// TIA Portal V17 export
// export: Created 2023-12-22T15:08:07.2930648Z, ExportSetting WithDefaults, DisplayName Totally Integrated Automation Portal, DisplayVersion V17, DisplayName TIA Portal Openness, DisplayVersion V17, DisplayName TIA Portal Version Control Interface, DisplayVersion V17, DisplayName STEP 7 Professional, DisplayVersion V17, DisplayName STEP 7 Safety, DisplayVersion V17, DisplayName WinCC Advanced, DisplayVersion V17
FUNCTION_BLOCK "Time_SYS"   // FB95, LAD
{ S7_Optimized_Access := 'FALSE' }
VERSION : 0.1
// stored: AutoNumber false, IsIECCheckEnabled false, SetENOAutomatically false, UDAEnableTagReadback false
   VAR DB_SPECIFIC
      Set_Time : Bool;   // Заданное время
      Time_Now : Struct   // Текущее время
         Year : Int;   // год
         Month : Int;   // месяц
         Day : Int;   // день месяца
         Weekday : Int;   // день недели (1 - воскресенье)
         Hour : Int;   // часы
         Minute : Int;   // минуты
         Second : Int;   // секунды
      END_STRUCT;
      Time_SP : Struct   // Текущее время
         Year : Int;   // год
         Month : Int;   // месяц
         Day : Int;   // день месяца
         Weekday : Int;   // день недели (1 - воскресенье)
         Hour : Int;   // часы
         Minute : Int;   // минуты
         Second : Int;   // секунды
      END_STRUCT;
      TimeZone { S7_SetPoint := 'True'} : TimeTransformationRule;   // Часовой пояс
      RD_SYS_Status : Int;   // Статус чтения времени
      WR_SYS_Status : Int;   // Статус записи времени
      RD_Time : DTL;   // Прочитанное сист. время
      SP_Time : DTL;   // Новое сист. время
   END_VAR
   VAR
      SET_TIMEZONE { S7_SetPoint := 'True'} : SET_TIMEZONE;   // Запись часового пояса
   END_VAR
   VAR DB_SPECIFIC
      Time_DTL : DTL;
   END_VAR
   // TimeZone.Bias := 180;   // Часовой пояс по GMT (смещение в минутах)
   // TimeZone.DaylightBias := 60;
   // TimeZone.DaylightStartMonth := 3;
   // TimeZone.DaylightStartWeek := 5;
   // TimeZone.DaylightStartWeekday := 7;
   // TimeZone.DaylightStartHour := 2;
   // TimeZone.DaylightStartMinute := 0;
   // TimeZone.StandardStartMonth := 10;
   // TimeZone.StandardStartWeek := 5;
   // TimeZone.StandardStartWeekday := 1;
   // TimeZone.StandardStartHour := 3;
   // TimeZone.StandardStartMinute := 0;
   // TimeZone.TimeZoneName := 'GMT+3';
   VAR_TEMP   // added for the SCL form of the ladder/FBD networks
      _w1 : Bool;
   END_VAR
BEGIN

REGION Network 1: Чтение системного времени
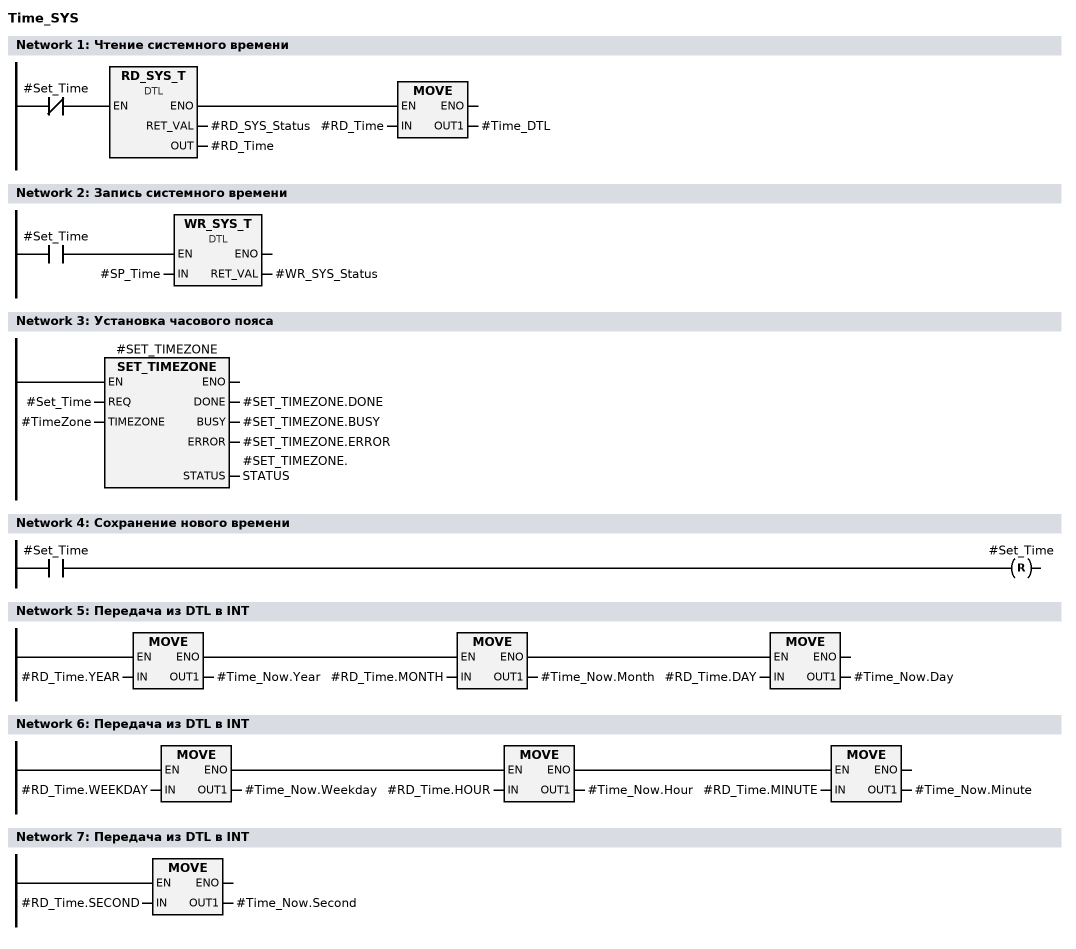
   RUNG wire#powerrail
      I_Contact( #Set_Time )
      { S7_Templates := "date_type := DTL" } RD_SYS_T(RET_VAL => #RD_SYS_Status, OUT => #RD_Time)
      Move(in := #RD_Time, out1 => #Time_DTL)
   END_RUNG
   // the same network as SCL:
   #RD_SYS_Status := RD_SYS_T(EN := NOT #Set_Time, OUT => #RD_Time, ENO => #_w1);
   IF #_w1 THEN #Time_DTL := #RD_Time; END_IF;
END_REGION

REGION Network 2: Запись системного времени
   RUNG wire#powerrail
      Contact( #Set_Time )
      { S7_Templates := "date_type := DTL" } WR_SYS_T(IN := #SP_Time, RET_VAL => #WR_SYS_Status)
   END_RUNG
   // the same network as SCL:
   IF #Set_Time THEN #WR_SYS_Status := WR_SYS_T(IN := #SP_Time); END_IF;
END_REGION

REGION Network 3: Установка часового пояса
   RUNG wire#powerrail
      #SET_TIMEZONE.SET_TIMEZONE(REQ := #Set_Time, TimeZone := #TimeZone, DONE => #SET_TIMEZONE.DONE, BUSY => #SET_TIMEZONE.BUSY, ERROR => #SET_TIMEZONE.ERROR, STATUS => #SET_TIMEZONE.STATUS)
   END_RUNG
   // the same network as SCL:
   #SET_TIMEZONE(REQ := #Set_Time,   // SET_TIMEZONE
                 TimeZone := #TimeZone,
                 DONE => #SET_TIMEZONE.DONE,
                 BUSY => #SET_TIMEZONE.BUSY,
                 ERROR => #SET_TIMEZONE.ERROR,
                 STATUS => #SET_TIMEZONE.STATUS);
END_REGION

REGION Network 4: Сохранение нового времени
   RUNG wire#powerrail
      Contact( #Set_Time )
      R_Coil( #Set_Time )
   END_RUNG
   // the same network as SCL:
   IF #Set_Time THEN #Set_Time := FALSE; END_IF;
END_REGION

REGION Network 5: Передача из DTL в INT
   RUNG wire#powerrail
      Move(in := #RD_Time.YEAR, out1 => #Time_Now.Year)
      Move(in := #RD_Time.MONTH, out1 => #Time_Now.Month)
      Move(in := #RD_Time.DAY, out1 => #Time_Now.Day)
   END_RUNG
   // the same network as SCL:
   #Time_Now.Year := #RD_Time.YEAR;
   #Time_Now.Month := #RD_Time.MONTH;
   #Time_Now.Day := #RD_Time.DAY;
END_REGION

REGION Network 6: Передача из DTL в INT
   RUNG wire#powerrail
      Move(in := #RD_Time.WEEKDAY, out1 => #Time_Now.Weekday)
      Move(in := #RD_Time.HOUR, out1 => #Time_Now.Hour)
      Move(in := #RD_Time.MINUTE, out1 => #Time_Now.Minute)
   END_RUNG
   // the same network as SCL:
   #Time_Now.Weekday := #RD_Time.WEEKDAY;
   #Time_Now.Hour := #RD_Time.HOUR;
   #Time_Now.Minute := #RD_Time.MINUTE;
END_REGION

REGION Network 7: Передача из DTL в INT
   RUNG wire#powerrail
      Move(in := #RD_Time.SECOND, out1 => #Time_Now.Second)
   END_RUNG
   // the same network as SCL:
   #Time_Now.Second := #RD_Time.SECOND;
END_REGION
END_FUNCTION_BLOCK
